{attribute 'qualified_only'}
//{attribute 'strict'}
{attribute 'to_string'}
TYPE eVendorNameID_1 :
(	
	NoVendor := 		0,
	BR := 				1,
	Beckhoff := 		2,
	Elmo := 			3,
	ControlTechnique :=	4,
	Servotronics := 	5,
	Nidec :=			6,
	LAST		
)DINT;
END_TYPE

(* stored: Version 1.1.0.1, ProductVersion 3.1.4024.3
   DUT eVendorNameID_1: Id {a8edc98d-141c-486b-95a0-9a4ba0853a56} *)
